// TIA Portal V20 export
TYPE "typeEstopStatus"
// stored: Access Published, IsFailsafeCompliant true, Namespace Safety
   STRUCT
      mainOpEmoPressed : Bool;   // Zone 1 - Main OP E-stop button is pressed
      unWinderLeftEmoPressed : Bool;   // Zone 1 - Unwinder E-stop button is pressed
      cutterEmoPressed : Bool;   // Zone 1 - Cutter E-stop button is pressed
      magazineEmoPressed : Bool;   // Zone 1 - Magazine E-stop button is pressed
      conveyorEmoPressed : Bool;   // Zone 1 - Conveyor E-stop button is pressed
      pHmi1EmoPressed : Bool;   // Zone 1 - PHMI1 E-stop button is pressed
      pHmi2EmoPressed : Bool;   // Zone 1 - PHMI2 E-stop button is pressed
      ba30EmoPressed : Bool;   // BA30 - E-stop button is pressed
      ba40EmoPressed : Bool;   // BA40 - E-stop button is pressed
      ba15EmoPressed : Bool;   // BA15 - E-stop button is pressed
      ba60EmoPressed : Bool;   // BA60 - E-stop button is pressed
   END_STRUCT;
END_TYPE
